// TIA Portal V18 export
// export: Created 2025-12-01T17:51:05.9540544Z, ExportSetting None, DisplayName Totally Integrated Automation Portal, DisplayVersion V18 Update 5, DisplayName TIA Portal Openness, DisplayVersion V18 Update 5, DisplayName TIA Portal Teamcenter Gateway, DisplayVersion V18, DisplayName TIA Portal Version Control Interface, DisplayVersion V18, DisplayName STEP 7 Professional, DisplayVersion V18 Update 5, DisplayName STEP 7 Safety, DisplayVersion V18, DisplayName WinCC Professional, DisplayVersion V18 Update 5
FUNCTION "ST10Cyl_interface91-100" : Void   // FC1029, LAD
{ S7_Optimized_Access := 'FALSE' }
// stored: AutoNumber false, SetENOAutomatically false
   VAR_INPUT
      AlwaysON : Bool;
      E_stop : Bool;
   END_VAR
   VAR_TEMP
      tTest : Bool;
   END_VAR
BEGIN

REGION Network 1 (SCL): Cylinder 91-100 IO Interface (SCL)
END_REGION

REGION Network 2: CY91 interface
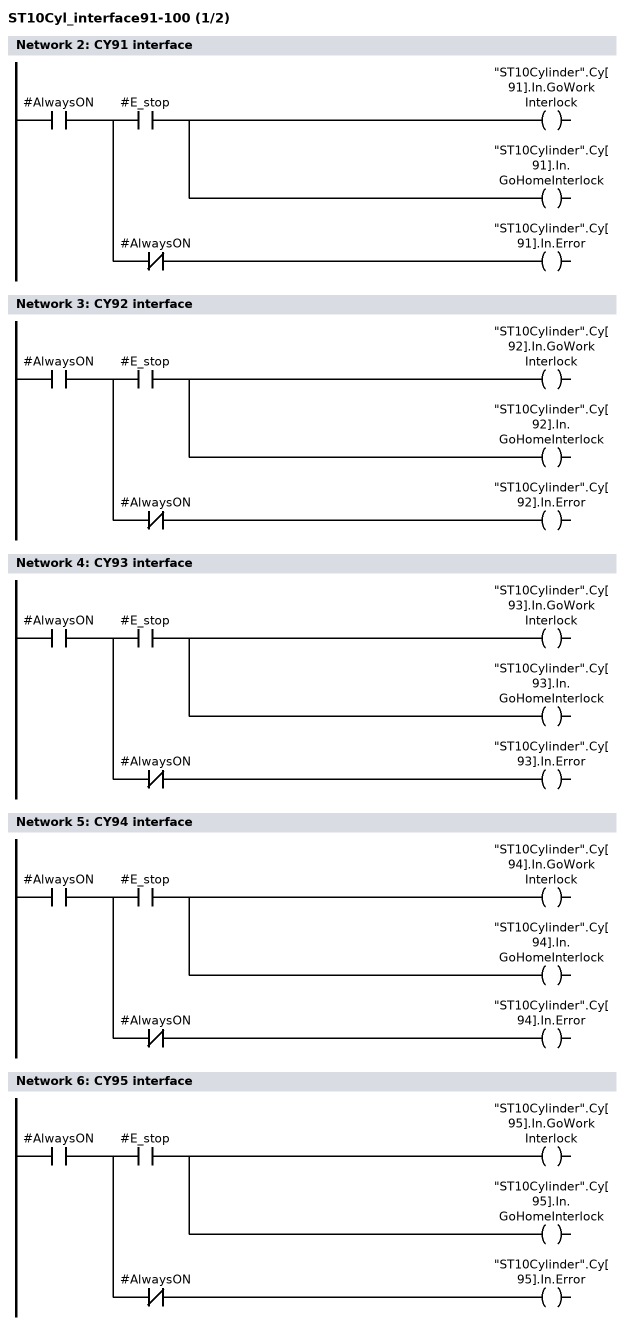
   RUNG wire#powerrail
      Contact( #AlwaysON )
      wire#w1
      Contact( #E_stop )
      wire#w2
      Coil( "ST10Cylinder".Cy[91].In.GoWorkInterlock )
   END_RUNG
   RUNG wire#w2
      Coil( "ST10Cylinder".Cy[91].In.GoHomeInterlock )
   END_RUNG
   RUNG wire#w1
      I_Contact( #AlwaysON )
      Coil( "ST10Cylinder".Cy[91].In.Error )
   END_RUNG
   // the same network as SCL:
   "ST10Cylinder".Cy[91].In.GoWorkInterlock := #AlwaysON AND #E_stop;
   "ST10Cylinder".Cy[91].In.GoHomeInterlock := #AlwaysON AND #E_stop;
   "ST10Cylinder".Cy[91].In.Error := #AlwaysON AND NOT #AlwaysON;
END_REGION

REGION Network 3: CY92 interface
   RUNG wire#powerrail
      Contact( #AlwaysON )
      wire#w1
      Contact( #E_stop )
      wire#w2
      Coil( "ST10Cylinder".Cy[92].In.GoWorkInterlock )
   END_RUNG
   RUNG wire#w2
      Coil( "ST10Cylinder".Cy[92].In.GoHomeInterlock )
   END_RUNG
   RUNG wire#w1
      I_Contact( #AlwaysON )
      Coil( "ST10Cylinder".Cy[92].In.Error )
   END_RUNG
   // the same network as SCL:
   "ST10Cylinder".Cy[92].In.GoWorkInterlock := #AlwaysON AND #E_stop;
   "ST10Cylinder".Cy[92].In.GoHomeInterlock := #AlwaysON AND #E_stop;
   "ST10Cylinder".Cy[92].In.Error := #AlwaysON AND NOT #AlwaysON;
END_REGION

REGION Network 4: CY93 interface
   RUNG wire#powerrail
      Contact( #AlwaysON )
      wire#w1
      Contact( #E_stop )
      wire#w2
      Coil( "ST10Cylinder".Cy[93].In.GoWorkInterlock )
   END_RUNG
   RUNG wire#w2
      Coil( "ST10Cylinder".Cy[93].In.GoHomeInterlock )
   END_RUNG
   RUNG wire#w1
      I_Contact( #AlwaysON )
      Coil( "ST10Cylinder".Cy[93].In.Error )
   END_RUNG
   // the same network as SCL:
   "ST10Cylinder".Cy[93].In.GoWorkInterlock := #AlwaysON AND #E_stop;
   "ST10Cylinder".Cy[93].In.GoHomeInterlock := #AlwaysON AND #E_stop;
   "ST10Cylinder".Cy[93].In.Error := #AlwaysON AND NOT #AlwaysON;
END_REGION

REGION Network 5: CY94 interface
   RUNG wire#powerrail
      Contact( #AlwaysON )
      wire#w1
      Contact( #E_stop )
      wire#w2
      Coil( "ST10Cylinder".Cy[94].In.GoWorkInterlock )
   END_RUNG
   RUNG wire#w2
      Coil( "ST10Cylinder".Cy[94].In.GoHomeInterlock )
   END_RUNG
   RUNG wire#w1
      I_Contact( #AlwaysON )
      Coil( "ST10Cylinder".Cy[94].In.Error )
   END_RUNG
   // the same network as SCL:
   "ST10Cylinder".Cy[94].In.GoWorkInterlock := #AlwaysON AND #E_stop;
   "ST10Cylinder".Cy[94].In.GoHomeInterlock := #AlwaysON AND #E_stop;
   "ST10Cylinder".Cy[94].In.Error := #AlwaysON AND NOT #AlwaysON;
END_REGION

REGION Network 6: CY95 interface
   RUNG wire#powerrail
      Contact( #AlwaysON )
      wire#w1
      Contact( #E_stop )
      wire#w2
      Coil( "ST10Cylinder".Cy[95].In.GoWorkInterlock )
   END_RUNG
   RUNG wire#w2
      Coil( "ST10Cylinder".Cy[95].In.GoHomeInterlock )
   END_RUNG
   RUNG wire#w1
      I_Contact( #AlwaysON )
      Coil( "ST10Cylinder".Cy[95].In.Error )
   END_RUNG
   // the same network as SCL:
   "ST10Cylinder".Cy[95].In.GoWorkInterlock := #AlwaysON AND #E_stop;
   "ST10Cylinder".Cy[95].In.GoHomeInterlock := #AlwaysON AND #E_stop;
   "ST10Cylinder".Cy[95].In.Error := #AlwaysON AND NOT #AlwaysON;
END_REGION

REGION Network 7: CY96 interface
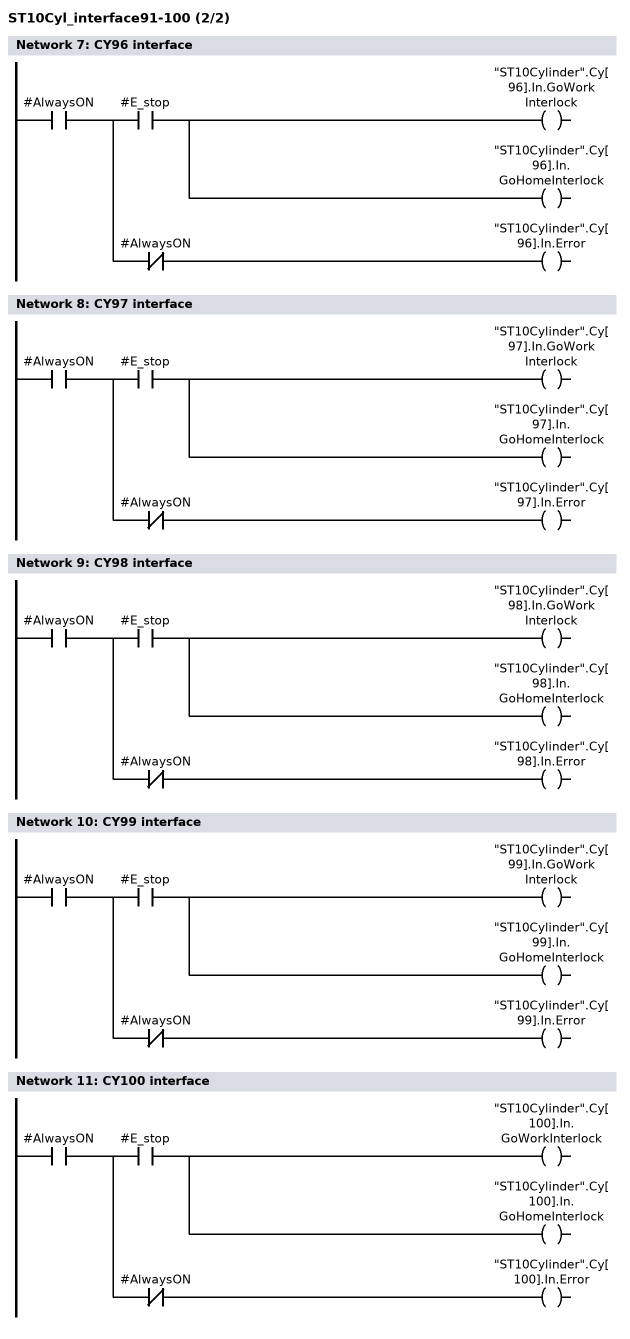
   RUNG wire#powerrail
      Contact( #AlwaysON )
      wire#w1
      Contact( #E_stop )
      wire#w2
      Coil( "ST10Cylinder".Cy[96].In.GoWorkInterlock )
   END_RUNG
   RUNG wire#w2
      Coil( "ST10Cylinder".Cy[96].In.GoHomeInterlock )
   END_RUNG
   RUNG wire#w1
      I_Contact( #AlwaysON )
      Coil( "ST10Cylinder".Cy[96].In.Error )
   END_RUNG
   // the same network as SCL:
   "ST10Cylinder".Cy[96].In.GoWorkInterlock := #AlwaysON AND #E_stop;
   "ST10Cylinder".Cy[96].In.GoHomeInterlock := #AlwaysON AND #E_stop;
   "ST10Cylinder".Cy[96].In.Error := #AlwaysON AND NOT #AlwaysON;
END_REGION

REGION Network 8: CY97 interface
   RUNG wire#powerrail
      Contact( #AlwaysON )
      wire#w1
      Contact( #E_stop )
      wire#w2
      Coil( "ST10Cylinder".Cy[97].In.GoWorkInterlock )
   END_RUNG
   RUNG wire#w2
      Coil( "ST10Cylinder".Cy[97].In.GoHomeInterlock )
   END_RUNG
   RUNG wire#w1
      I_Contact( #AlwaysON )
      Coil( "ST10Cylinder".Cy[97].In.Error )
   END_RUNG
   // the same network as SCL:
   "ST10Cylinder".Cy[97].In.GoWorkInterlock := #AlwaysON AND #E_stop;
   "ST10Cylinder".Cy[97].In.GoHomeInterlock := #AlwaysON AND #E_stop;
   "ST10Cylinder".Cy[97].In.Error := #AlwaysON AND NOT #AlwaysON;
END_REGION

REGION Network 9: CY98 interface
   RUNG wire#powerrail
      Contact( #AlwaysON )
      wire#w1
      Contact( #E_stop )
      wire#w2
      Coil( "ST10Cylinder".Cy[98].In.GoWorkInterlock )
   END_RUNG
   RUNG wire#w2
      Coil( "ST10Cylinder".Cy[98].In.GoHomeInterlock )
   END_RUNG
   RUNG wire#w1
      I_Contact( #AlwaysON )
      Coil( "ST10Cylinder".Cy[98].In.Error )
   END_RUNG
   // the same network as SCL:
   "ST10Cylinder".Cy[98].In.GoWorkInterlock := #AlwaysON AND #E_stop;
   "ST10Cylinder".Cy[98].In.GoHomeInterlock := #AlwaysON AND #E_stop;
   "ST10Cylinder".Cy[98].In.Error := #AlwaysON AND NOT #AlwaysON;
END_REGION

REGION Network 10: CY99 interface
   RUNG wire#powerrail
      Contact( #AlwaysON )
      wire#w1
      Contact( #E_stop )
      wire#w2
      Coil( "ST10Cylinder".Cy[99].In.GoWorkInterlock )
   END_RUNG
   RUNG wire#w2
      Coil( "ST10Cylinder".Cy[99].In.GoHomeInterlock )
   END_RUNG
   RUNG wire#w1
      I_Contact( #AlwaysON )
      Coil( "ST10Cylinder".Cy[99].In.Error )
   END_RUNG
   // the same network as SCL:
   "ST10Cylinder".Cy[99].In.GoWorkInterlock := #AlwaysON AND #E_stop;
   "ST10Cylinder".Cy[99].In.GoHomeInterlock := #AlwaysON AND #E_stop;
   "ST10Cylinder".Cy[99].In.Error := #AlwaysON AND NOT #AlwaysON;
END_REGION

REGION Network 11: CY100 interface
   RUNG wire#powerrail
      Contact( #AlwaysON )
      wire#w1
      Contact( #E_stop )
      wire#w2
      Coil( "ST10Cylinder".Cy[100].In.GoWorkInterlock )
   END_RUNG
   RUNG wire#w2
      Coil( "ST10Cylinder".Cy[100].In.GoHomeInterlock )
   END_RUNG
   RUNG wire#w1
      I_Contact( #AlwaysON )
      Coil( "ST10Cylinder".Cy[100].In.Error )
   END_RUNG
   // the same network as SCL:
   "ST10Cylinder".Cy[100].In.GoWorkInterlock := #AlwaysON AND #E_stop;
   "ST10Cylinder".Cy[100].In.GoHomeInterlock := #AlwaysON AND #E_stop;
   "ST10Cylinder".Cy[100].In.Error := #AlwaysON AND NOT #AlwaysON;
END_REGION
END_FUNCTION
